Staubli VAL3: iPlate2.pgx

public program iPlate2(num& nNum[] (dimensions=1))
begin
  nNum=dioGet(iPlate2)
end
